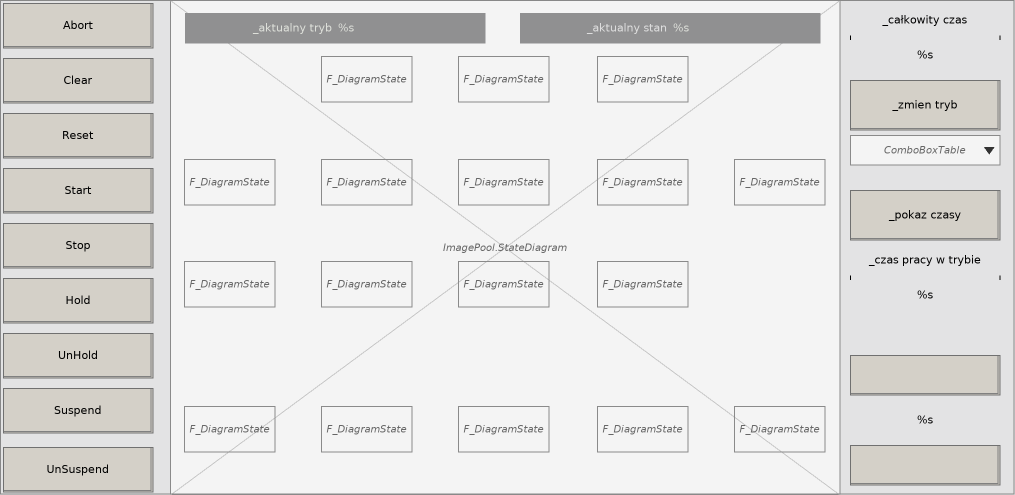
VISUALIZATION F_06_Diagram  // 1015x495
VAR_IN_OUT
	stScreenData	: ST_MCHMIPrepareScreen_06_XX;
	
END_VAR
    Rectangle (850,5 150x65)
    Image (170,0 670x495), image: ImagePool.StateDiagram
    Rectangle (185,13 150x30), "_aktualny tryb", text list: 'TextListGlobal', text index: 1
    Rectangle (335,13 150x30), "%s", text variable: stScreenData.wsActualMode
    Rectangle (520,13 150x30), "_aktualny stan", text list: 'TextListGlobal', text index: 0
    Rectangle (670,13 150x30), "%s", text variable: stScreenData.wsActualState
    Frame (734,406 91x46), invisible if: not stScreenData.arrStateEnabledInMode [1]
        shows F_DiagramState(stStateInfo := stScreenData.arrState [1])
    Frame (597,406 91x46), invisible if: not stScreenData.arrStateEnabledInMode [2]
        shows F_DiagramState(stStateInfo := stScreenData.arrState [2])
    Frame (458,406 91x46), invisible if: not stScreenData.arrStateEnabledInMode [3]
        shows F_DiagramState(stStateInfo := stScreenData.arrState [3])
    Frame (321,406 91x46), invisible if: not stScreenData.arrStateEnabledInMode [4]
        shows F_DiagramState(stStateInfo := stScreenData.arrState [4])
    Frame (184,406 91x46), invisible if: not stScreenData.arrStateEnabledInMode [5]
        shows F_DiagramState(stStateInfo := stScreenData.arrState [5])
    Frame (597,261 91x46), invisible if: not stScreenData.arrStateEnabledInMode [10]
        shows F_DiagramState(stStateInfo := stScreenData.arrState [10])
    Frame (458,261 91x46), invisible if: not stScreenData.arrStateEnabledInMode [11]
        shows F_DiagramState(stStateInfo := stScreenData.arrState [11])
    Frame (321,261 91x46), invisible if: not stScreenData.arrStateEnabledInMode [12]
        shows F_DiagramState(stStateInfo := stScreenData.arrState [12])
    Frame (184,261 91x46), invisible if: not stScreenData.arrStateEnabledInMode [6]
        shows F_DiagramState(stStateInfo := stScreenData.arrState [6])
    Frame (734,159 91x46), invisible if: not stScreenData.arrStateEnabledInMode [17]
        shows F_DiagramState(stStateInfo := stScreenData.arrState [17])
    Frame (597,159 91x46), invisible if: not stScreenData.arrStateEnabledInMode [16]
        shows F_DiagramState(stStateInfo := stScreenData.arrState [16])
    Frame (458,159 91x46), invisible if: not stScreenData.arrStateEnabledInMode [9]
        shows F_DiagramState(stStateInfo := stScreenData.arrState [9])
    Frame (321,159 91x46), invisible if: not stScreenData.arrStateEnabledInMode [8]
        shows F_DiagramState(stStateInfo := stScreenData.arrState [8])
    Frame (184,159 91x46), invisible if: not stScreenData.arrStateEnabledInMode [7]
        shows F_DiagramState(stStateInfo := stScreenData.arrState [7])
    Frame (597,56 91x46), invisible if: not stScreenData.arrStateEnabledInMode [13]
        shows F_DiagramState(stStateInfo := stScreenData.arrState [13])
    Frame (458,56 91x46), invisible if: not stScreenData.arrStateEnabledInMode [14]
        shows F_DiagramState(stStateInfo := stScreenData.arrState [14])
    Frame (321,56 91x46), invisible if: not stScreenData.arrStateEnabledInMode [15]
        shows F_DiagramState(stStateInfo := stScreenData.arrState [15])
    Button (3,58 150x45), "Clear", text list: 'TextList_Opisy'
        OnMouseDown: execute { stScreenData.arrCmdChangeState [E_SaMCommandChangeState.Clear].bPushed := true; }
    Button (3,113 150x45), "Reset", text list: 'TextList_Opisy'
        OnMouseDown: execute { stScreenData.arrCmdChangeState [E_SaMCommandChangeState.Reset].bPushed := true; }
    Button (3,168 150x45), "Start", text list: 'TextList_Opisy'
        OnMouseDown: execute { stScreenData.arrCmdChangeState [E_SaMCommandChangeState.Start].bPushed := true; }
    Button (3,388 150x45), "Suspend", text list: 'TextList_Opisy'
        OnMouseDown: execute { stScreenData.arrCmdChangeState [E_SaMCommandChangeState.Suspend].bPushed := true; }
    Button (3,447 150x45), "UnSuspend", text list: 'TextList_Opisy'
        OnMouseDown: execute { stScreenData.arrCmdChangeState [E_SaMCommandChangeState.Unsuspend].bPushed := true; }
    Button (3,278 150x45), "Hold", text list: 'TextList_Opisy'
        OnMouseDown: execute { stScreenData.arrCmdChangeState [E_SaMCommandChangeState.Hold].bPushed := true; }
    Button (3,333 150x45), "UnHold", text list: 'TextList_Opisy'
        OnMouseDown: execute { stScreenData.arrCmdChangeState [E_SaMCommandChangeState.Unhold].bPushed := true; }
    Button (3,3 150x45), "Abort"
        OnMouseDown: execute { stScreenData.arrCmdChangeState [E_SaMCommandChangeState.Abort ].bPushed := true; }
    Button (3,223 150x45), "Stop", text list: 'TextList_Opisy'
        OnMouseDown: execute { stScreenData.arrCmdChangeState [E_SaMCommandChangeState.Stop].bPushed := true; }
    Rectangle (850,5 150x30), "_całkowity czas", text list: 'TextList_06', text index: 0
    Rectangle (850,40 150x30), "%s", text variable: stScreenData.sTotalWorkTime
    Button (850,80 150x50), "_zmien tryb", text list: 'TextList_06', text index: 1
        OnMouseDown: execute { stScreenData.bChangeMode := TRUE; }
    Button (850,190 150x50), "_pokaz czasy", text list: 'TextList_06', text index: 2
        toggle stScreenData.bShowTime
    Rectangle (850,245 150x65), invisible if: not stScreenData.bShowTime
    Rectangle (850,245 150x30), "_czas pracy w trybie", invisible if: not stScreenData.bShowTime, text list: 'TextList_06', text index: 3
    Rectangle (850,280 150x30), "%s", text variable: stScreenData.sWorkingTimeInMode, invisible if: not stScreenData.bShowTime
    ComboBoxTable (850,135 150x30), variable: stScreenData.iSelectedMode, data array: stScreenData.arrNamesOfMode
        p3854506369: stScreenData.arrNamesOfMode[INDEX].wsDescription
        p1892666644: stScreenData.arrNamesOfMode[INDEX].iNumber
    Button (850,355 150x40), invisible if: not stScreenData.bShowTime, text list: 'TextList_06', text index: 4
        OnMouseDown: execute { stScreenData.bNextModeToDisplayTime := TRUE; }
    Button (850,445 150x40), invisible if: not stScreenData.bShowTime, text list: 'TextList_06', text index: 5
        OnMouseDown: execute { stScreenData.bPrevModeToDisplayTime := TRUE; }
    Rectangle (850,405 150x30), "%s", text variable: stScreenData.wsNameModeOfTimeDisplay, invisible if: not stScreenData.bShowTime
END_VISUALIZATION

(* stored: Version 1.1.0.1
   Visu F_06_Diagram: Id {b5a56d21-7772-0579-081c-3efd13b48022} *)
